// TIA Portal V18 program export: 0 tag tables, 0 data types, 0 data blocks, 1 code blocks (in call order from the OBs), 0 instance data blocks

ORGANIZATION_BLOCK "Main"   // OB1, FBD, ProgramCycle
TITLE = "Main Program Sweep (Cycle)"
{ S7_Optimized_Access := 'TRUE' }
VERSION : 0.1
// stored: AutoNumber true, IsIECCheckEnabled false, SetENOAutomatically false
   VAR_INPUT
      Initial_Call : Bool;   // Initial call of this OB
      Remanence : Bool;   // =True, if remanent data are available
   END_VAR
   VAR_TEMP
      MB_PORT_SET_OK : Bool;
   END_VAR
BEGIN

REGION Network 2 (SCL)
   //Leak Test FC
   // "Leak_Test"(InOUT := "Data_SEQ".CYL_Leak_Test);
   "Data_SEQ".CYL_Leak_Test_L.Timer.PT:= DINT_TO_TIME(INT_TO_DINT("Data_SEQ".CYL_Leak_Test_L.Duration_Set) * 1000 * 60);
   "Data_SEQ".DECAY_Leak_Test_L.Timer.PT := DINT_TO_TIME(INT_TO_DINT("Data_SEQ".DECAY_Leak_Test_L.Duration_Set) * 1000 * 60);
   "Data_SEQ".V3_Leak_Test_L.Timer.PT := DINT_TO_TIME(INT_TO_DINT("Data_SEQ".V3_Leak_Test_L.Duration_Set) * 1000 * 60);
   "Data_SEQ".HP_Leak_Test_L.Timer.PT := DINT_TO_TIME(INT_TO_DINT("Data_SEQ".HP_Leak_Test_L.Duration_Set) * 1000 * 60);
   "Data_SEQ".Stable_Leak_Test_L.Timer.PT := DINT_TO_TIME(INT_TO_DINT("Data_SEQ".Stable_Leak_Test_L.Duration_Set) * 1000 * 60);

   //Leak Test FC
   // "Leak_Test"(InOUT := "Data_SEQ".CYL_Leak_Test);
   "Data_SEQ".CYL_Leak_Test_R.Timer.PT := DINT_TO_TIME(INT_TO_DINT("Data_SEQ".CYL_Leak_Test_R.Duration_Set) * 1000 * 60);
   "Data_SEQ".DECAY_Leak_Test_R.Timer.PT := DINT_TO_TIME(INT_TO_DINT("Data_SEQ".DECAY_Leak_Test_R.Duration_Set) * 1000 * 60);
   "Data_SEQ".V3_Leak_Test_R.Timer.PT := DINT_TO_TIME(INT_TO_DINT("Data_SEQ".V3_Leak_Test_R.Duration_Set) * 1000 * 60);
   "Data_SEQ".HP_Leak_Test_R.Timer.PT := DINT_TO_TIME(INT_TO_DINT("Data_SEQ".HP_Leak_Test_R.Duration_Set) * 1000 * 60);
   "Data_SEQ".Stable_Leak_Test_R.Timer.PT := DINT_TO_TIME(INT_TO_DINT("Data_SEQ".Stable_Leak_Test_R.Duration_Set) * 1000 * 60);


   //Purge Heater Timer 55555
   "Countdown_Timer"(Start_bit:="Data_MODBUS_PID"."Pre-Heater Time".Start,
                     Duration_Set:="Data_MODBUS_PID"."Pre-Heater Time".Duration_Set,
                     "timer":="Data_MODBUS_PID"."Pre-Heater Time".Timer,
                     Display_Hr:="Data_MODBUS_PID"."Pre-Heater Time".Display_time.Hr,
                     Display_Min:="Data_MODBUS_PID"."Pre-Heater Time".Display_time.Min,
                     Display_Sec:="Data_MODBUS_PID"."Pre-Heater Time".Display_time.Sec);
END_REGION

REGION Network 3 (SCL): 193
   "HMI_OP_DB"();

   "Password_Login_DB"();

   "Netmap_mapping_DB"();
   "IP_Change_DB"();
   "ARS_Connect"();
   "To_ARS_Sign_DB"();


   //Intial option
   "Initail setup and Option code_DB"();


   //Mapping
   "Data_Mapping_DB"();

   //Operator
   "SEQ_PREM_DB"();
   "SEQ_OPERATOR_DB"();

   "Reset_DB"();

   //SEQ//L
   "IDL_L_DB"();

   "Pre_Purge_L_DB"();

   "Change_Cyl_L_DB"();



   "PostPruge_L_DB"();

   "Rough_Line_L_DB"();

   "PanelPurge_L_DB"();

   "Proc_Gas_L_DB"();



   //SEQ//R
   "IDL_R_DB"();


   "PanelPurge_R_DB"();


   "Pre_Purge_R_DB"();
   "Change_Cyl_R_DB"();
   "PostPruge_R_DB"();
   "Rough_Line_R_DB"();


   "Proc_Gas_R_DB"();





   //Sub SEQ//L
   "HP_SIDE_L_DB"();
   "Cond_Cycle_L_DB"();
   "LP_SIDE_L_DB"();
   "LP_Panel_L_DB"();
   "Outboard_L_DB"();


   //Sub SEQ//R
   "Cond_Cycle_R_DB"();
   "HP_SIDE_R_DB"();
   "LP_Panel_R_DB"();
   "LP_SIDE_R_DB"();
   "Outboard_R_DB"();






   //Barcode and Cyclinder EXP
   "Barcode_Type_In_DB"();
   "Expiration Date_all_DB"();




   //DO
   "Valve_Output_DB"();
   "Relay_Defaults_DB"();


   //Alarm
   "Alarm_Output_DB"();
   "AL_Resp_SEQ_and_Flag_DB"();

   //AI
   "Analog_Alarm_DB"();

   //DI
   "DI_IntFlg_IntAlm_Alarm_DB"();


   // IF "Data_ModBusData"."MB[760].8_Total_Shutdown_Alarm_#1" OR "Data_ModBusData"."MB[760].9_Total_Shutdown_Alarm_#2"
   //     OR "Data_ModBusData"."MB[760].10_Total_Shutdown_Alarm_#3" OR "Data_ModBusData"."MB[760].11_Total_Shutdown_Alarm_#4"
   // THEN
   //     "Data_ModBusData"."MB[534]_Prompt_INFO" := 0;
   //     "Data_ModBusData"."MB[800].0_Prompt_Common_Comfirm" := FALSE;
   //     "Data_ModBusData"."MB[800].1_Prompt_Common_On" := FALSE;
   // END_IF;
   // 
   "First_SetIP_Delay".TON(IN:="First_SetIP_Delay_Bit",
                           PT:=T#3s);


   REGION First Set IP
       // Statement section REGION

       IF "RDREC_DATA_DB".RDREC_M0[20] = 0 AND "First_SetIP_Delay".Q
       THEN
           "First_IP_Assign" := true;
           "Main_PLC_To_ARS_Connection_DB".RemoteAddress.ADDR[1] := 19;
           "Main_PLC_To_ARS_Connection_DB".RemoteAddress.ADDR[2] := 19;
           "Main_PLC_To_ARS_Connection_DB".RemoteAddress.ADDR[3] := 19;
           "Main_PLC_To_ARS_Connection_DB".RemoteAddress.ADDR[4] := 11;
           "First_SetIP_Delay_Bit" := false;
       END_IF;

   END_REGION



   //*****Start up, 延後Alarm開始掃描時間*****//
   IF "Alarm_Delay_ON" = TRUE
   THEN
       "PW ON_Alarm delay" := TRUE;
       // RESET_TIMER("IEC_Timer_PW ON_Alarm delay");
   END_IF;


   "IEC_Timer_0_DB_4".TON(IN := NOT "Alarm_Delay_ON",
                          PT := T#1S);


   IF "IEC_Timer_0_DB_4".Q
   THEN
       "Alarm_Delay_ON" := TRUE;
   END_IF;

   "IEC_Timer_PW ON_Alarm delay".TON(IN:="PW ON_Alarm delay",
                                     PT:=T#10S);



   REGION watchDog
       "WatchDog_Counter".CTU(CU := "Watch_Dog",
                              PV := 5);
       "IEC_Timer_0_DB_2".TON(IN := "Watch_Dog",
                              PT := T#1S);

       "IEC_Timer_0_DB_3".TON(IN:="Watch_Dog2",
                              PT:=T#1S);

       IF "IEC_Timer_0_DB_2".Q = FALSE
       THEN
           "Watch_Dog2" := TRUE;
       ELSE
           "Watch_Dog" := FALSE;

       END_IF;

       IF "IEC_Timer_0_DB_3".Q = FALSE
       THEN
           "Watch_Dog" := TRUE;
       ELSE
           "Watch_Dog2" := FALSE;

       END_IF;

       IF "WatchDog_Counter".QU
       THEN
           "WatchDog_Counter".R := 1;

       END_IF;

       IF "WatchDog_Counter".CV = 1
       THEN
           "WatchDog_Counter".R := 0;
           "Data_Netmap".Data[24] := 20;
       ELSIF "WatchDog_Counter".CV = 2
       THEN
           "Data_Netmap".Data[24] := 40;
       ELSIF "WatchDog_Counter".CV = 3
       THEN
           "Data_Netmap".Data[24] := 60;
       ELSIF "WatchDog_Counter".CV = 4
       THEN
           "Data_Netmap".Data[24] := 80;
       ELSIF "WatchDog_Counter".CV = 5
       THEN
           "Data_Netmap".Data[24] := 100;

       END_IF;

       IF "WatchDog_Counter".CV > 5
       THEN
           "WatchDog_Counter".CV := 0;
       END_IF;

   END_REGION

   REGION I/O ERROR
       // Statement section REGION

       "Data_Error data".retvalue := ModuleStates(LADDR := "Data_Error data".LADDR, MODE := "Data_Error data".MODE, STATE := "Data_Error data".state);
       IF "Data_Error data"."IO Error TEST_bypass" = FALSE
       THEN
           "Data_Internal_Flag_and_Alarm"."IAlarm[5]_I/O_ERROR".Trigger := "Data_Error data".state[0];
       ELSE
           "Data_Internal_Flag_and_Alarm"."IAlarm[5]_I/O_ERROR".Trigger := FALSE;
       END_IF;

       // "Data_Internal_Flag_and_Alarm"."IAlarm[5]_I/O_ERROR".Enable_1 := TRUE;
       // "Data_Internal_Flag_and_Alarm"."IAlarm[5]_I/O_ERROR".Enable_3 := TRUE;

   END_REGION
END_REGION
END_ORGANIZATION_BLOCK
